// TIA Portal project "SLMP" (V20)

(* hardware
DEVICE "S7-1500/ET200MP station_1"  S7-1500 station
   slot 0: "Rail_0"  Rack  6ES7 590-1***0-0AA0
   slot 1: "PLC_1"  CPU 1516F-3 PN/DP  6ES7 516-3FN01-0AB0  V2.9
      slot 3: "CPU display_1"  6ES7591-1BA00-0AA0
      slot 32768: "PROFINET interface_1"  X1
      slot 33024: "PROFINET interface_2"  X2
      slot 33280: "DP interface_1"  X3
      slot 34817: "Virtual CP interface port_1"  Virtual CP interface port  Virtual CP interface port
*)

// ===== PLC "PLC_1"  CPU 1516F-3 PN/DP =====

VAR_GLOBAL   // PLC tag table "Default tag table"
   "Tag_1" AT %MD100 : UDInt;
   "Tag_2" AT %MB200 : Byte;
   "Tag_3" AT %MB201 : Byte;
   "Tag_4" AT %MB202 : Byte;
   "Tag_5" AT %MB203 : Byte;
END_VAR

TYPE "udtSLMPDeviceCode"
   STRUCT
      D : Bool;
      "M" : Bool;
      X : Bool;
      Y : Bool;
      W : Bool;
   END_STRUCT;
END_TYPE

DATA_BLOCK "dbFX5Read"   // DB1
{ S7_Optimized_Access := 'TRUE' }
VERSION : 0.1
   VAR
      arrb : Array[0..1024] of Byte;
      udtTCON_IP_v4 : TCON_IP_v4;
      xStart : Bool;
      xStop : Bool;
      xReset : Bool;
      xAutoReset : Bool;
   END_VAR
   VAR RETAIN
      uiFirstDeviceOffset : UInt;
      uiTotalDevices : UInt;
      udtSLMPDeviceCode : "udtSLMPDeviceCode";
   END_VAR
   VAR
      xBusy : Bool;
      xError : Bool;
      uiDoneCount : UInt;
      uiErrorCount : UInt;
      iErrorID : Int;
      iCurrentStep : Int;
   END_VAR
BEGIN
END_DATA_BLOCK

DATA_BLOCK "fbCom2FX5_DB"   // DB2
{ S7_Optimized_Access := 'TRUE' }
VERSION : 0.1
// stored: InstanceOfName fbCom2FX5
"fbCom2FX5"
BEGIN
END_DATA_BLOCK

DATA_BLOCK "dbFX5Write"   // DB3
{ S7_Optimized_Access := 'TRUE' }
VERSION : 0.1
   VAR
      arrb : Array[0..1024] of Byte;
      udtTCON_IP_v4 : TCON_IP_v4;
      xStart : Bool;
      xStop : Bool;
      xReset : Bool;
      xAutoReset : Bool;
   END_VAR
   VAR RETAIN
      uiFirstDeviceOffset : UInt;
      uiTotalDevices : UInt;
      udtSLMPDeviceCode : "udtSLMPDeviceCode";
   END_VAR
   VAR
      xBusy : Bool;
      xError : Bool;
      uiDoneCount : UInt;
      uiErrorCount : UInt;
      iErrorID : Int;
      iCurrentStep : Int;
   END_VAR
BEGIN
END_DATA_BLOCK

FUNCTION_BLOCK "fbSLMPRead"   // FB1, SCL
{ S7_Optimized_Access := 'TRUE' }
VERSION : 0.1
   VAR_INPUT
      xStart : Bool;
      xStop : Bool;
      xReset : Bool;
      xAutoReset : Bool;
      CONN_OUC : Conn_Ouc;
      uiFirstDeviceOffset : UInt;
      uiTotalDevices : UInt := 1;
      udtSLMPDeviceCode : "udtSLMPDeviceCode";
   END_VAR
   VAR_OUTPUT
      xBusy : Bool;
      xError : Bool;
      uiDoneCount : UInt;
      uiErrorCount : UInt;
      iErrorID : Int;
      iCurrentStep : Int;
   END_VAR
   VAR_IN_OUT
      udtTCON_IP_v4 : TCON_IP_v4;
      arrb : Array[0..#ebufferLength] of Byte;
   END_VAR
   VAR
      arrfbTONs : Array[0..1] of TON_TIME;
      fbTCON : TCON;
      fbTSEND : TSEND;
      fbTRCV : TRCV;
      fbTDISCON : TDISCON;
      iStep : Int;
      xTCONReq : Bool;
      xTSENDReq : Bool;
      xTRCVReq : Bool;
      xTDISReq : Bool;
      xCycleStop : Bool;
      arrbSendBuffer : Array[0..#ebufferLength] of Byte;
      arrbReceBuffer : Array[0..#ebufferLength] of Byte;
      fbR_TRIG : Array[0..5] of R_TRIG;
   END_VAR
   VAR_TEMP
      _uiLoop : UInt;
      _arrbTempArray : Array[0..3] of Byte;
   END_VAR
   VAR CONSTANT
      ebufferLength : UInt := 1024;
      e3EFrame : Byte := 16#50;
   END_VAR
BEGIN

   #fbR_TRIG[0](CLK := #xStart);
   #fbR_TRIG[1](CLK := #xStop AND #iStep > 0);
   IF #fbR_TRIG[1].Q THEN
       #xCycleStop := True;
   END_IF;

   CASE #iStep OF
       0:
           #xTCONReq := FALSE;
           #xTSENDReq := False;
           #xTRCVReq := false;
           #xTDISReq := False;
           #xCycleStop := False;
           #xError := FALSE;
           #xBusy := false;
           #arrfbTONs[0](IN := False,
                         PT := T#0.1s);
           #arrfbTONs[1](IN := False,
                         PT := T#0.1s);
           IF NOT #fbTCON.ERROR AND NOT #fbTCON.BUSY
               AND NOT #fbTDISCON.ERROR AND NOT #fbTDISCON.BUSY
               AND NOT #fbTSEND.ERROR AND NOT #fbTSEND.BUSY
               AND NOT #fbTCON.ERROR AND NOT #fbTCON.BUSY
               AND #fbR_TRIG[0].Q
           THEN
               FOR #_uiLoop := 0 TO #ebufferLength DO
                   #arrbSendBuffer[#_uiLoop] := 0;
                   #arrbReceBuffer[#_uiLoop] := 0;
               END_FOR;
               #xBusy := True;
               #iStep := 5;
           END_IF;
       5:
           IF NOT #udtSLMPDeviceCode.D
               AND NOT #udtSLMPDeviceCode.M
               AND NOT #udtSLMPDeviceCode.W
               AND NOT #udtSLMPDeviceCode.X
               AND NOT #udtSLMPDeviceCode.Y
           THEN
               #iStep := 9005;
               #iErrorID := 9005;
           ELSIF #uiTotalDevices <= 0 THEN
               #iStep := 9005;
               #iErrorID := 9005;
           ELSE
               #iStep := 10;
           END_IF;
       10:
           #arrfbTONs[0](IN := False,
                         PT := T#0.1s);
           #xTCONReq := True;
           IF #fbTCON.BUSY THEN
               #iStep := 15;
           END_IF;
       15:
           IF #fbTCON.STATUS=0 THEN
               #iStep := 20;
           END_IF;
       20:
           //50 00 00 ff ff 03 00 0c 00 10 00 01 04 00 00 64 00 00 a8 0a 00
           //0  1  2  3   4  5  6  7  8  9 10 11 12 13 14 15 16 17 18 19 20
           #arrbSendBuffer[0] := #e3EFrame;
           //
           #arrbSendBuffer[1] := 16#0;
           //Network Number
           #arrbSendBuffer[2] := 16#0;
           //SubNetwork Number
           #arrbSendBuffer[3] := 16#FF;
           //Requested unit I/O number
           #arrbSendBuffer[4] := 16#FF;
           #arrbSendBuffer[5] := 16#03;
           //Requesting Unit Station Number
           #arrbSendBuffer[6] := 16#00;
           //Requested data length Bytes
           #arrbSendBuffer[7] := 16#0C;
           #arrbSendBuffer[8] := 16#00;
           //Monitor Timer
           #arrbSendBuffer[9] := 16#10;
           #arrbSendBuffer[10] := 16#00;
           //Command
           #arrbSendBuffer[11] := 16#01;
           #arrbSendBuffer[12] := 16#04;
           //SubCommand
           #arrbSendBuffer[13] := 16#00;
           #arrbSendBuffer[14] := 16#00;

           // #arrbSendBuffer[15] := 16#64;
           // #arrbSendBuffer[16] := 16#00;
           // #arrbSendBuffer[17] := 16#00;
           // #arrbSendBuffer[18] := 16#A8;
           // #arrbSendBuffer[19] := 16#0A;
           // #arrbSendBuffer[20] := 16#00;

           //first number of Register
           "fc32BitDataTo4Bytes"(
                                 in := #uiFirstDeviceOffset,
                                 b0 => #arrbSendBuffer[15],
                                 b1 => #arrbSendBuffer[16],
                                 b2 => #arrbSendBuffer[17],
                                 b3 => #_arrbTempArray[0]
           );
           //device code
           #arrbSendBuffer[18] := "fcSLMPGetDeviceCode"(udtSLMPDeviceCode := #udtSLMPDeviceCode);
           //numbers
           "fc32BitDataTo4Bytes"(
                                 in := #uiTotalDevices,
                                 b0 => #arrbSendBuffer[19],
                                 b1 => #arrbSendBuffer[20],
                                 b2 => #_arrbTempArray[0],
                                 b3 => #_arrbTempArray[1]
           );
           #iStep := 30;
       30:
           #fbTSEND.LEN := 21;
           #xTSENDReq := True;
           IF #fbTSEND.BUSY THEN
               #iStep := 33;
           END_IF;
       33:
           #arrfbTONs[0](
                         IN := True,
                         PT := T#3s
           );
           IF #fbTSEND.STATUS=0 THEN
               #arrfbTONs[0](
                             IN := False,
                             PT := T#3s
               );
               #iStep := 35;
           END_IF;
           IF #arrfbTONs[0].Q THEN
               #iStep := 9033;
               #iErrorID := 9033;
           END_IF;
       35:
           #xTSENDReq := False;
           #xTRCVReq := True;
           #arrfbTONs[0](
                         IN := True,
                         PT := T#1s
           );
           IF #fbTRCV.RCVD_LEN > 0 THEN
               #arrfbTONs[0](
                             IN := False,
                             PT := T#3s
               );
               #iStep := 40;
           END_IF;
           IF #arrfbTONs[0].Q THEN
               #iStep := 9035;
               #iErrorID := 9035;
           END_IF;
       40:
           #xTRCVReq := false;
           IF NOT #fbTRCV.BUSY THEN
               #iStep := 50;
           END_IF;
       50:
           //IF arrbReceBuffer[0]
           IF #arrbReceBuffer[0] <> 16#D0 AND #arrbReceBuffer[9] <> 16#00 AND #arrbReceBuffer[10] <> 16#00 THEN
               #iStep := 9050;
               #iErrorID := 9050;
           ELSE
               #iStep := 60;
           END_IF;

       60:
           FOR #_uiLoop := 0 TO #ebufferLength-11 DO
               #arrb[#_uiLoop] := #arrbReceBuffer[#_uiLoop +11];
           END_FOR;

           #uiDoneCount := #uiDoneCount + 1;
           IF NOT #xCycleStop THEN

              #iStep := 70;

           ELSE
               #iStep := 100;
           END_IF;
       70:
           #iStep := 20;
       100:
           #xTDISReq := True;
           IF #fbTDISCON.BUSY THEN
               #iStep := 105;
           END_IF;
       105:
           IF  #xCycleStop THEN
               #iStep := 0;
           ELSE
               IF #xAutoReset THEN
                   #iStep := 0;
               ELSE
                   IF #xReset THEN
                       #iStep := 0;
                   END_IF;
               END_IF;
           END_IF;

       9005:
           #iStep := 0;
       9010..9999:
           #arrfbTONs[0](
                         IN := False,
                         PT := T#3s
           );
           #xError := True;
           #iStep := 100;

   END_CASE;

   #fbR_TRIG[2](CLK := #xError);
   IF #fbR_TRIG[2].Q THEN
       #uiErrorCount := #uiErrorCount + 1;
   END_IF;

   #iCurrentStep := #iStep;


   #fbTCON(
           REQ:=#xTCONReq,
           ID:=#CONN_OUC,
           CONNECT:=#udtTCON_IP_v4
   );

   #fbTDISCON(
              ID := #CONN_OUC,
              REQ := #xTDISReq
   );

   #fbTSEND(
            ID := #CONN_OUC,
            REQ := #xTSENDReq,
            DATA := #arrbSendBuffer
   );

   #fbTRCV(
           ID := #CONN_OUC,
           EN_R := #xTRCVReq,
           LEN:=0,
           ADHOC:=True,
           DATA := #arrbReceBuffer

   );
END_FUNCTION_BLOCK

FUNCTION_BLOCK "fbCom2FX5"   // FB2, LAD
{ S7_Optimized_Access := 'TRUE' }
VERSION : 0.1
   VAR
      fbSLMPRead_Instance : "fbSLMPRead";
      fbSLMPWrite : "fbSLMPWrite";
   END_VAR
   VAR_TEMP
      _xOut : Bool;
   END_VAR
BEGIN

REGION Network 1: ReadData via SLMP
END_REGION

REGION Network 2: ..Remote IP Address
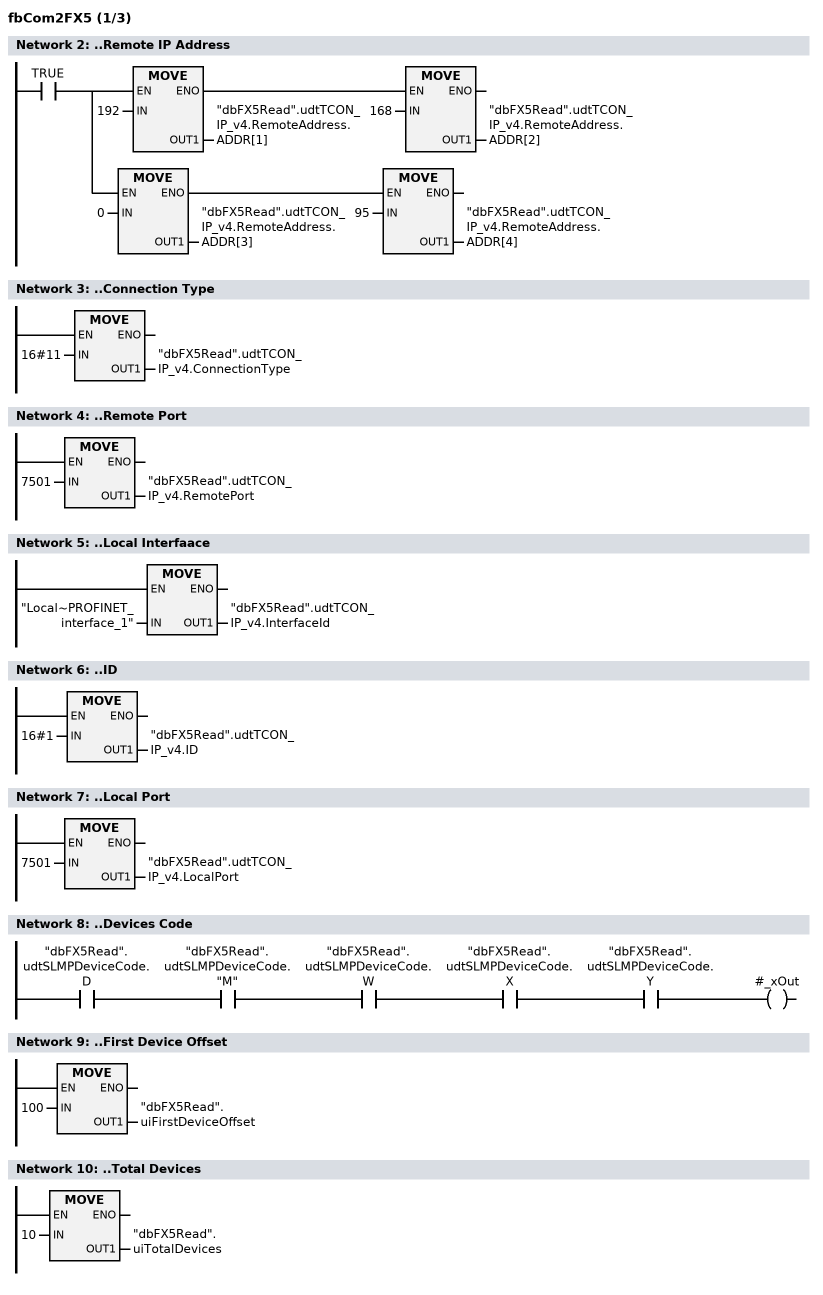
   RUNG wire#powerrail
      Contact( TRUE )
      wire#w1
      Move(in := 192, out1 => "dbFX5Read".udtTCON_IP_v4.RemoteAddress.ADDR[1])
      Move(in := 168, out1 => "dbFX5Read".udtTCON_IP_v4.RemoteAddress.ADDR[2])
   END_RUNG
   RUNG wire#w1
      Move(in := 0, out1 => "dbFX5Read".udtTCON_IP_v4.RemoteAddress.ADDR[3])
      Move(in := 95, out1 => "dbFX5Read".udtTCON_IP_v4.RemoteAddress.ADDR[4])
   END_RUNG
   // the same network as SCL:
   IF TRUE THEN
       "dbFX5Read".udtTCON_IP_v4.RemoteAddress.ADDR[1] := 192;
       "dbFX5Read".udtTCON_IP_v4.RemoteAddress.ADDR[2] := 168;
       "dbFX5Read".udtTCON_IP_v4.RemoteAddress.ADDR[3] := 0;
       "dbFX5Read".udtTCON_IP_v4.RemoteAddress.ADDR[4] := 95;
   END_IF;
END_REGION

REGION Network 3: ..Connection Type
   RUNG wire#powerrail
      Move(in := 16#11, out1 => "dbFX5Read".udtTCON_IP_v4.ConnectionType)
   END_RUNG
   // the same network as SCL:
   "dbFX5Read".udtTCON_IP_v4.ConnectionType := 16#11;
END_REGION

REGION Network 4: ..Remote Port
   RUNG wire#powerrail
      Move(in := 7501, out1 => "dbFX5Read".udtTCON_IP_v4.RemotePort)
   END_RUNG
   // the same network as SCL:
   "dbFX5Read".udtTCON_IP_v4.RemotePort := 7501;
END_REGION

REGION Network 5: ..Local Interfaace
   RUNG wire#powerrail
      Move(in := "Local~PROFINET_interface_1", out1 => "dbFX5Read".udtTCON_IP_v4.InterfaceId)
   END_RUNG
   // the same network as SCL:
   "dbFX5Read".udtTCON_IP_v4.InterfaceId := "Local~PROFINET_interface_1";
END_REGION

REGION Network 6: ..ID
   RUNG wire#powerrail
      Move(in := 16#1, out1 => "dbFX5Read".udtTCON_IP_v4.ID)
   END_RUNG
   // the same network as SCL:
   "dbFX5Read".udtTCON_IP_v4.ID := 16#1;
END_REGION

REGION Network 7: ..Local Port
   RUNG wire#powerrail
      Move(in := 7501, out1 => "dbFX5Read".udtTCON_IP_v4.LocalPort)
   END_RUNG
   // the same network as SCL:
   "dbFX5Read".udtTCON_IP_v4.LocalPort := 7501;
END_REGION

REGION Network 8: ..Devices Code
   RUNG wire#powerrail
      Contact( "dbFX5Read".udtSLMPDeviceCode.D )
      Contact( "dbFX5Read".udtSLMPDeviceCode."M" )
      Contact( "dbFX5Read".udtSLMPDeviceCode.W )
      Contact( "dbFX5Read".udtSLMPDeviceCode.X )
      Contact( "dbFX5Read".udtSLMPDeviceCode.Y )
      Coil( #_xOut )
   END_RUNG
   // the same network as SCL:
   #_xOut := "dbFX5Read".udtSLMPDeviceCode.D AND "dbFX5Read".udtSLMPDeviceCode."M" AND "dbFX5Read".udtSLMPDeviceCode.W AND "dbFX5Read".udtSLMPDeviceCode.X AND "dbFX5Read".udtSLMPDeviceCode.Y;
END_REGION

REGION Network 9: ..First Device Offset
   RUNG wire#powerrail
      Move(in := 100, out1 => "dbFX5Read".uiFirstDeviceOffset)
   END_RUNG
   // the same network as SCL:
   "dbFX5Read".uiFirstDeviceOffset := 100;
END_REGION

REGION Network 10: ..Total Devices
   RUNG wire#powerrail
      Move(in := 10, out1 => "dbFX5Read".uiTotalDevices)
   END_RUNG
   // the same network as SCL:
   "dbFX5Read".uiTotalDevices := 10;
END_REGION

REGION Network 11: ..active/passive connection establishment
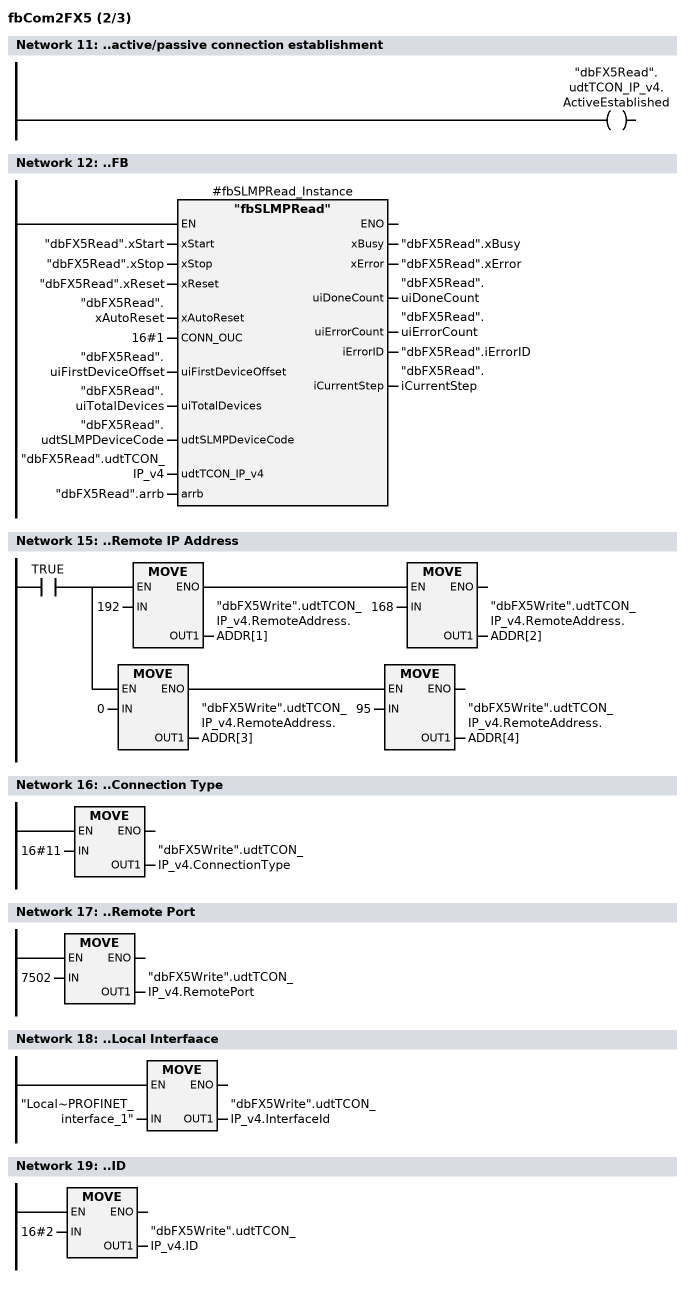
   RUNG wire#powerrail
      Coil( "dbFX5Read".udtTCON_IP_v4.ActiveEstablished )
   END_RUNG
   // the same network as SCL:
   "dbFX5Read".udtTCON_IP_v4.ActiveEstablished := TRUE;
END_REGION

REGION Network 12: ..FB
   RUNG wire#powerrail
      #fbSLMPRead_Instance(xStart := "dbFX5Read".xStart, xStop := "dbFX5Read".xStop, xReset := "dbFX5Read".xReset, xAutoReset := "dbFX5Read".xAutoReset, CONN_OUC := 16#1, uiFirstDeviceOffset := "dbFX5Read".uiFirstDeviceOffset, uiTotalDevices := "dbFX5Read".uiTotalDevices, udtSLMPDeviceCode := "dbFX5Read".udtSLMPDeviceCode, udtTCON_IP_v4 := "dbFX5Read".udtTCON_IP_v4, arrb := "dbFX5Read".arrb, xBusy => "dbFX5Read".xBusy, xError => "dbFX5Read".xError, uiDoneCount => "dbFX5Read".uiDoneCount, uiErrorCount => "dbFX5Read".uiErrorCount, iErrorID => "dbFX5Read".iErrorID, iCurrentStep => "dbFX5Read".iCurrentStep)
   END_RUNG
   // the same network as SCL:
   #fbSLMPRead_Instance(xStart := "dbFX5Read".xStart,   // "fbSLMPRead"
                        xStop := "dbFX5Read".xStop,
                        xReset := "dbFX5Read".xReset,
                        xAutoReset := "dbFX5Read".xAutoReset,
                        CONN_OUC := 16#1,
                        uiFirstDeviceOffset := "dbFX5Read".uiFirstDeviceOffset,
                        uiTotalDevices := "dbFX5Read".uiTotalDevices,
                        udtSLMPDeviceCode := "dbFX5Read".udtSLMPDeviceCode,
                        udtTCON_IP_v4 := "dbFX5Read".udtTCON_IP_v4,
                        arrb := "dbFX5Read".arrb,
                        xBusy => "dbFX5Read".xBusy,
                        xError => "dbFX5Read".xError,
                        uiDoneCount => "dbFX5Read".uiDoneCount,
                        uiErrorCount => "dbFX5Read".uiErrorCount,
                        iErrorID => "dbFX5Read".iErrorID,
                        iCurrentStep => "dbFX5Read".iCurrentStep);
END_REGION

REGION Network 13: WriteData via SLMP
END_REGION

REGION Network 15: ..Remote IP Address
   RUNG wire#powerrail
      Contact( TRUE )
      wire#w1
      Move(in := 192, out1 => "dbFX5Write".udtTCON_IP_v4.RemoteAddress.ADDR[1])
      Move(in := 168, out1 => "dbFX5Write".udtTCON_IP_v4.RemoteAddress.ADDR[2])
   END_RUNG
   RUNG wire#w1
      Move(in := 0, out1 => "dbFX5Write".udtTCON_IP_v4.RemoteAddress.ADDR[3])
      Move(in := 95, out1 => "dbFX5Write".udtTCON_IP_v4.RemoteAddress.ADDR[4])
   END_RUNG
   // the same network as SCL:
   IF TRUE THEN
       "dbFX5Write".udtTCON_IP_v4.RemoteAddress.ADDR[1] := 192;
       "dbFX5Write".udtTCON_IP_v4.RemoteAddress.ADDR[2] := 168;
       "dbFX5Write".udtTCON_IP_v4.RemoteAddress.ADDR[3] := 0;
       "dbFX5Write".udtTCON_IP_v4.RemoteAddress.ADDR[4] := 95;
   END_IF;
END_REGION

REGION Network 16: ..Connection Type
   RUNG wire#powerrail
      Move(in := 16#11, out1 => "dbFX5Write".udtTCON_IP_v4.ConnectionType)
   END_RUNG
   // the same network as SCL:
   "dbFX5Write".udtTCON_IP_v4.ConnectionType := 16#11;
END_REGION

REGION Network 17: ..Remote Port
   RUNG wire#powerrail
      Move(in := 7502, out1 => "dbFX5Write".udtTCON_IP_v4.RemotePort)
   END_RUNG
   // the same network as SCL:
   "dbFX5Write".udtTCON_IP_v4.RemotePort := 7502;
END_REGION

REGION Network 18: ..Local Interfaace
   RUNG wire#powerrail
      Move(in := "Local~PROFINET_interface_1", out1 => "dbFX5Write".udtTCON_IP_v4.InterfaceId)
   END_RUNG
   // the same network as SCL:
   "dbFX5Write".udtTCON_IP_v4.InterfaceId := "Local~PROFINET_interface_1";
END_REGION

REGION Network 19: ..ID
   RUNG wire#powerrail
      Move(in := 16#2, out1 => "dbFX5Write".udtTCON_IP_v4.ID)
   END_RUNG
   // the same network as SCL:
   "dbFX5Write".udtTCON_IP_v4.ID := 16#2;
END_REGION

REGION Network 20: ..Local Port
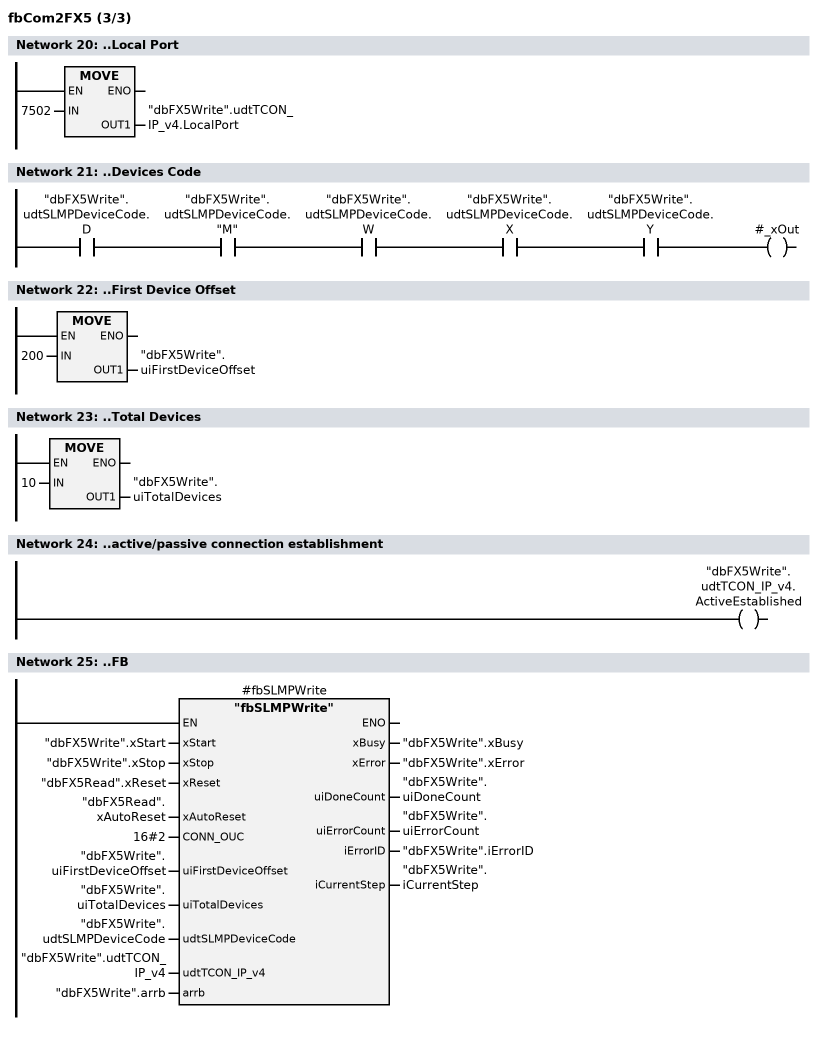
   RUNG wire#powerrail
      Move(in := 7502, out1 => "dbFX5Write".udtTCON_IP_v4.LocalPort)
   END_RUNG
   // the same network as SCL:
   "dbFX5Write".udtTCON_IP_v4.LocalPort := 7502;
END_REGION

REGION Network 21: ..Devices Code
   RUNG wire#powerrail
      Contact( "dbFX5Write".udtSLMPDeviceCode.D )
      Contact( "dbFX5Write".udtSLMPDeviceCode."M" )
      Contact( "dbFX5Write".udtSLMPDeviceCode.W )
      Contact( "dbFX5Write".udtSLMPDeviceCode.X )
      Contact( "dbFX5Write".udtSLMPDeviceCode.Y )
      Coil( #_xOut )
   END_RUNG
   // the same network as SCL:
   #_xOut := "dbFX5Write".udtSLMPDeviceCode.D AND "dbFX5Write".udtSLMPDeviceCode."M" AND "dbFX5Write".udtSLMPDeviceCode.W AND "dbFX5Write".udtSLMPDeviceCode.X AND "dbFX5Write".udtSLMPDeviceCode.Y;
END_REGION

REGION Network 22: ..First Device Offset
   RUNG wire#powerrail
      Move(in := 200, out1 => "dbFX5Write".uiFirstDeviceOffset)
   END_RUNG
   // the same network as SCL:
   "dbFX5Write".uiFirstDeviceOffset := 200;
END_REGION

REGION Network 23: ..Total Devices
   RUNG wire#powerrail
      Move(in := 10, out1 => "dbFX5Write".uiTotalDevices)
   END_RUNG
   // the same network as SCL:
   "dbFX5Write".uiTotalDevices := 10;
END_REGION

REGION Network 24: ..active/passive connection establishment
   RUNG wire#powerrail
      Coil( "dbFX5Write".udtTCON_IP_v4.ActiveEstablished )
   END_RUNG
   // the same network as SCL:
   "dbFX5Write".udtTCON_IP_v4.ActiveEstablished := TRUE;
END_REGION

REGION Network 25: ..FB
   RUNG wire#powerrail
      #fbSLMPWrite(xStart := "dbFX5Write".xStart, xStop := "dbFX5Write".xStop, xReset := "dbFX5Read".xReset, xAutoReset := "dbFX5Read".xAutoReset, CONN_OUC := 16#2, uiFirstDeviceOffset := "dbFX5Write".uiFirstDeviceOffset, uiTotalDevices := "dbFX5Write".uiTotalDevices, udtSLMPDeviceCode := "dbFX5Write".udtSLMPDeviceCode, udtTCON_IP_v4 := "dbFX5Write".udtTCON_IP_v4, arrb := "dbFX5Write".arrb, xBusy => "dbFX5Write".xBusy, xError => "dbFX5Write".xError, uiDoneCount => "dbFX5Write".uiDoneCount, uiErrorCount => "dbFX5Write".uiErrorCount, iErrorID => "dbFX5Write".iErrorID, iCurrentStep => "dbFX5Write".iCurrentStep)
   END_RUNG
   // the same network as SCL:
   #fbSLMPWrite(xStart := "dbFX5Write".xStart,   // "fbSLMPWrite"
                xStop := "dbFX5Write".xStop,
                xReset := "dbFX5Read".xReset,
                xAutoReset := "dbFX5Read".xAutoReset,
                CONN_OUC := 16#2,
                uiFirstDeviceOffset := "dbFX5Write".uiFirstDeviceOffset,
                uiTotalDevices := "dbFX5Write".uiTotalDevices,
                udtSLMPDeviceCode := "dbFX5Write".udtSLMPDeviceCode,
                udtTCON_IP_v4 := "dbFX5Write".udtTCON_IP_v4,
                arrb := "dbFX5Write".arrb,
                xBusy => "dbFX5Write".xBusy,
                xError => "dbFX5Write".xError,
                uiDoneCount => "dbFX5Write".uiDoneCount,
                uiErrorCount => "dbFX5Write".uiErrorCount,
                iErrorID => "dbFX5Write".iErrorID,
                iCurrentStep => "dbFX5Write".iCurrentStep);
END_REGION
END_FUNCTION_BLOCK

FUNCTION_BLOCK "fbSLMPWrite"   // FB3, SCL
{ S7_Optimized_Access := 'TRUE' }
VERSION : 0.1
   VAR_INPUT
      xStart : Bool;
      xStop : Bool;
      xReset : Bool;
      xAutoReset : Bool;
      CONN_OUC : Conn_Ouc;
      uiFirstDeviceOffset : UInt;
      uiTotalDevices : UInt := 1;
      udtSLMPDeviceCode : "udtSLMPDeviceCode";
   END_VAR
   VAR_OUTPUT
      xBusy : Bool;
      xError : Bool;
      uiDoneCount : UInt;
      uiErrorCount : UInt;
      iErrorID : Int;
      iCurrentStep : Int;
   END_VAR
   VAR_IN_OUT
      udtTCON_IP_v4 : TCON_IP_v4;
      arrb : Array[0..#ebufferLength] of Byte;
   END_VAR
   VAR
      arrfbTONs : Array[0..1] of TON_TIME;
      fbTCON : TCON;
      fbTSEND : TSEND;
      fbTRCV : TRCV;
      fbTDISCON : TDISCON;
      iStep : Int;
      xTCONReq : Bool;
      xTSENDReq : Bool;
      xTRCVReq : Bool;
      xTDISReq : Bool;
      xCycleStop : Bool;
      arrbSendBuffer : Array[0..#ebufferLength] of Byte;
      arrbReceBuffer : Array[0..#ebufferLength] of Byte;
      fbR_TRIG : Array[0..5] of R_TRIG;
   END_VAR
   VAR_TEMP
      _uiLoop : UInt;
      _uiSendDataTotalLength : UInt;
      _arrbTempArray : Array[0..3] of Byte;
   END_VAR
   VAR CONSTANT
      ebufferLength : UInt := 1024;
      e3EFrame : Byte := 16#50;
   END_VAR
BEGIN

   #fbR_TRIG[0](CLK := #xStart);
   #fbR_TRIG[1](CLK := #xStop AND #iStep > 0);
   IF #fbR_TRIG[1].Q THEN
       #xCycleStop := True;
   END_IF;

   CASE #iStep OF
       0:
           #xTCONReq := FALSE;
           #xTSENDReq := False;
           #xTRCVReq := false;
           #xTDISReq := False;
           #xCycleStop := False;
           #xError := FALSE;
           #xBusy := false;
           #arrfbTONs[0](IN := False,
                         PT := T#0.1s);
           #arrfbTONs[1](IN := False,
                         PT := T#0.1s);
           IF NOT #fbTCON.ERROR AND NOT #fbTCON.BUSY
               AND NOT #fbTDISCON.ERROR AND NOT #fbTDISCON.BUSY
               AND NOT #fbTSEND.ERROR AND NOT #fbTSEND.BUSY
               AND NOT #fbTCON.ERROR AND NOT #fbTCON.BUSY
               AND #fbR_TRIG[0].Q
           THEN
               FOR #_uiLoop := 0 TO #ebufferLength DO
                   #arrbSendBuffer[#_uiLoop] := 0;
                   #arrbReceBuffer[#_uiLoop] := 0;
               END_FOR;
               #xBusy := True;
               #iStep := 5;
           END_IF;
       5:
           IF NOT #udtSLMPDeviceCode.D
               AND NOT #udtSLMPDeviceCode.M
               AND NOT #udtSLMPDeviceCode.W
               AND NOT #udtSLMPDeviceCode.X
               AND NOT #udtSLMPDeviceCode.Y
           THEN
               #iStep := 9005;
               #iErrorID := 9005;
           ELSIF #uiTotalDevices <= 0 THEN
               #iStep := 9005;
               #iErrorID := 9005;
           ELSE
               #iStep := 10;
           END_IF;
       10:
           #arrfbTONs[0](IN := False,
                         PT := T#0.1s);
           #xTCONReq := True;
           IF #fbTCON.BUSY THEN
               #iStep := 15;
           END_IF;
       15:
           IF #fbTCON.STATUS = 0 THEN
               #iStep := 20;
           END_IF;
       20:
           //50 00 00 ff ff 03 00 0c 00 10 00 01 04 00 00 64 00 00 a8 0a 00
           //0  1  2  3   4  5  6  7  8  9 10 11 12 13 14 15 16 17 18 19 20
           #arrbSendBuffer[0] := #e3EFrame;
           //
           #arrbSendBuffer[1] := 16#0;
           //Network Number
           #arrbSendBuffer[2] := 16#0;
           //SubNetwork Number
           #arrbSendBuffer[3] := 16#FF;
           //Requested unit I/O number
           #arrbSendBuffer[4] := 16#FF;
           #arrbSendBuffer[5] := 16#03;
           //Requesting Unit Station Number
           #arrbSendBuffer[6] := 16#00;
           //Requested data length Bytes
           #_uiSendDataTotalLength := #uiTotalDevices * 2 + 12;
           "fc32BitDataTo4Bytes"(
                                 in := #_uiSendDataTotalLength,
                                 b0 => #_arrbTempArray[0],
                                 b1 => #_arrbTempArray[1],
                                 b2 => #_arrbTempArray[2],
                                 b3 => #_arrbTempArray[3]
           );
           #arrbSendBuffer[7] := #_arrbTempArray[0];
           #arrbSendBuffer[8] := #_arrbTempArray[1];
           //Monitor Timer
           #arrbSendBuffer[9] := 16#10;
           #arrbSendBuffer[10] := 16#00;
           //Command
           #arrbSendBuffer[11] := 16#01;
           #arrbSendBuffer[12] := 16#14;
           //SubCommand
           #arrbSendBuffer[13] := 16#00;
           #arrbSendBuffer[14] := 16#00;

           //first number of Register
           "fc32BitDataTo4Bytes"(
                                 in := #uiFirstDeviceOffset,
                                 b0 => #arrbSendBuffer[15],
                                 b1 => #arrbSendBuffer[16],
                                 b2 => #arrbSendBuffer[17],
                                 b3 => #_arrbTempArray[0]
           );
           //device code
           #arrbSendBuffer[18] := "fcSLMPGetDeviceCode"(udtSLMPDeviceCode := #udtSLMPDeviceCode);
           //numbers
           "fc32BitDataTo4Bytes"(
                                 in := #uiTotalDevices,
                                 b0 => #arrbSendBuffer[19],
                                 b1 => #arrbSendBuffer[20],
                                 b2 => #_arrbTempArray[0],
                                 b3 => #_arrbTempArray[1]
           );

           FOR #_uiLoop := 0 TO #ebufferLength-21 DO
               #arrbSendBuffer[21 + #_uiLoop] := #arrb[#_uiLoop];
           END_FOR;
           #iStep := 30;
           ;
       30:
           #fbTSEND.LEN := 21 + #uiTotalDevices * 2;;
           #xTSENDReq := True;
           IF #fbTSEND.BUSY THEN
               #iStep := 33;
           END_IF;
       33:
           #arrfbTONs[0](
                         IN := True,
                         PT := T#3s
           );
           IF #fbTSEND.STATUS = 0 THEN
               #arrfbTONs[0](
                             IN := False,
                             PT := T#3s
               );
               #iStep := 35;
           END_IF;
           IF #arrfbTONs[0].Q THEN
               #iStep := 9033;
               #iErrorID := 9033;
           END_IF;
       35:
           #xTSENDReq := False;
           #xTRCVReq := True;
           #arrfbTONs[0](
                         IN := True,
                         PT := T#1s
           );
           IF #fbTRCV.RCVD_LEN > 0 THEN
               #arrfbTONs[0](
                             IN := False,
                             PT := T#3s
               );
               #iStep := 40;
           END_IF;
           IF #arrfbTONs[0].Q THEN
               #iStep := 9035;
               #iErrorID := 9035;
           END_IF;
       40:
           #xTRCVReq := false;
           IF NOT #fbTRCV.BUSY THEN
               #iStep := 50;
           END_IF;
       50:
           //IF arrbReceBuffer[0]
           IF #arrbReceBuffer[0] <> 16#D0 AND #arrbReceBuffer[9] <> 16#00 AND #arrbReceBuffer[10] <> 16#00 THEN
               #iStep := 9050;
               #iErrorID := 9050;
           ELSE
               #iStep := 60;
           END_IF;

       60:
           //#arrb := #arrbReceBuffer;
           #uiDoneCount := #uiDoneCount + 1;
           IF NOT #xCycleStop THEN

               #iStep := 70;

           ELSE
               #iStep := 100;
           END_IF;
       70:
           #iStep := 20;
       100:
           #xTDISReq := True;
           IF #fbTDISCON.BUSY THEN
               #iStep := 105;
           END_IF;
       105:
           IF #xCycleStop THEN
               #iStep := 0;
           ELSE
               IF #xAutoReset THEN
                   #iStep := 0;
               ELSE
                   IF #xReset THEN
                       #iStep := 0;
                   END_IF;
               END_IF;
           END_IF;
       9005:
           #iStep := 0;
       9010..9999:
           #arrfbTONs[0](
                         IN := False,
                         PT := T#3s
           );
           #xError := True;
           #iStep := 100;

   END_CASE;

   #fbR_TRIG[2](CLK := #xError);
   IF #fbR_TRIG[2].Q THEN
       #uiErrorCount := #uiErrorCount + 1;
   END_IF;

   #iCurrentStep := #iStep;


   #fbTCON(
           REQ := #xTCONReq,
           ID := #CONN_OUC,
           CONNECT := #udtTCON_IP_v4
   );

   #fbTDISCON(
              ID := #CONN_OUC,
              REQ := #xTDISReq
   );

   #fbTSEND(
            ID := #CONN_OUC,
            REQ := #xTSENDReq,
            DATA := #arrbSendBuffer
   );

   #fbTRCV(
           ID := #CONN_OUC,
           EN_R := #xTRCVReq,
           LEN := 0,
           ADHOC := True,
           DATA := #arrbReceBuffer

   );
END_FUNCTION_BLOCK

FUNCTION "fcSLMPGetDeviceCode" : Byte   // FC1, SCL
{ S7_Optimized_Access := 'TRUE' }
VERSION : 0.1
   VAR_INPUT
      udtSLMPDeviceCode : "udtSLMPDeviceCode";
   END_VAR
   VAR CONSTANT
      eDeviceCodeD : Byte := 16#A8;
      eDeviceCodeM : Byte := 16#90;
      eDeviceCodeX : Byte := 16#9C;
      eDeviceCodeY : Byte := 16#9D;
      eDeviceCodeW : Byte := 16#B4;
   END_VAR
BEGIN
   #fcSLMPGetDeviceCode := 16#0;

   IF #udtSLMPDeviceCode.D THEN
       #fcSLMPGetDeviceCode := #eDeviceCodeD;
   ELSIF #udtSLMPDeviceCode.M THEN
       #fcSLMPGetDeviceCode := #eDeviceCodeM;
   ELSIF #udtSLMPDeviceCode.W THEN
       #fcSLMPGetDeviceCode := #eDeviceCodeW;
   ELSIF #udtSLMPDeviceCode.X THEN
       #fcSLMPGetDeviceCode := #eDeviceCodeX;
   ELSIF #udtSLMPDeviceCode.Y THEN
       #fcSLMPGetDeviceCode := #eDeviceCodeY;
   END_IF;
END_FUNCTION

FUNCTION "fc32BitDataTo4Bytes" : Void   // FC2, SCL
{ S7_Optimized_Access := 'TRUE' }
VERSION : 0.1
   VAR_INPUT
      in : UDInt;
   END_VAR
   VAR_OUTPUT
      b0 : Byte;
      b1 : Byte;
      b2 : Byte;
      b3 : Byte;
   END_VAR
BEGIN
   #b0 := #in.%B0;
   #b1 := #in.%B1;
   #b2 := #in.%B2;
   #b3 := #in.%B3;
END_FUNCTION

ORGANIZATION_BLOCK "Main"   // OB1, LAD, ProgramCycle
TITLE = "Main Program Sweep (Cycle)"
{ S7_Optimized_Access := 'TRUE' }
VERSION : 0.1
   VAR_INPUT
      Initial_Call : Bool;   // Initial call of this OB
      Remanence : Bool;   // =True, if remanent data are available
   END_VAR
BEGIN

REGION Network 2
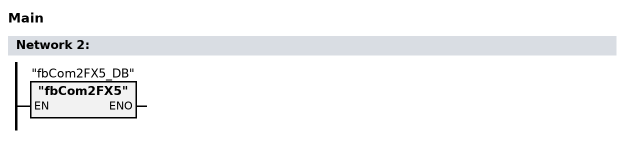
   RUNG wire#powerrail
      "fbCom2FX5_DB"()
   END_RUNG
   // the same network as SCL:
   "fbCom2FX5_DB"();   // "fbCom2FX5"
END_REGION
END_ORGANIZATION_BLOCK